// TIA Portal V20 export
DATA_BLOCK "DB_OPC_Recipe"   // DB134
{ S7_Optimized_Access := 'TRUE' }
// stored: MemoryReserve 100
   VAR RETAIN
      Current : Struct
         RecipeId : DInt;
         RecipeVersionGuid : String;
      END_STRUCT;
   END_VAR
   VAR
      Data : Struct
         LaserJobListName : String;
         RecipeId : DInt;
         RecipeName : String;
         RecipeVersionGuid : String;
         Station1 : Struct
            General : Struct
               Detections : Struct
                  WorkPart : Struct
                     Max : LReal;
                     Min : LReal;
                  END_STRUCT;
               END_STRUCT;
               GazPressure : Struct
                  WorkLaserDefault : LReal;
               END_STRUCT;
            END_STRUCT;
         END_STRUCT;
      END_STRUCT;
      TransferToPlc : Bool;
   END_VAR
BEGIN
END_DATA_BLOCK
